// TwinCAT 3 PLC project main
// ProgramVersion: 3.1.4024.0
// libraries:
//   Tc2_Standard, * (Beckhoff Automation GmbH)
//   Tc2_System, * (Beckhoff Automation GmbH)
//   Tc3_Module, * (Beckhoff Automation GmbH)
// project tree:
//   DUTs/ SafeState.TcDUT
//   GVLs/ IO.TcGVL
//   / PlcTask.TcTTO
//   POUs/ FB_EdgeDetector.TcPOU, MAIN.TcPOU
// real-time tasks:
//   TASK PlcTask: cycle T#10ms, priority 20, ADS port 350
// I/O:
//   DEVICE Device 1 (EtherCAT), AmsNetId 10.180.42.11.2.1
//     Term 1 (EK1200) [EK1200-5000 EtherCAT Power supply (2A E-Bus)]
//       Term 2 (EL1004) [EL1004 4Ch. Dig. Input 24V, 3ms]
//       Term 3 (EL2004) [EL2004 4Ch. Dig. Output 24V, 0.5A]
//       Term 4 (EL3004) [EL3004 4Ch. Ana. Input +/-10V]
//       Term 5 (EL4034) [EL4034 4Ch. Ana. Output +/-10V, 12bit]
//       Term 6 (EK1110) [EK1110 EtherCAT extension]
// variable links:
//   main/main Instance <-> Device 1 (EtherCAT)/Term 1 (EK1200)/Term 2 (EL1004)
//     PlcTask Inputs/IO.bBlueButton <-> Channel 2/Input
//     PlcTask Inputs/IO.bYellowButton <-> Channel 1/Input
//   main/main Instance <-> Device 1 (EtherCAT)/Term 1 (EK1200)/Term 3 (EL2004)
//     PlcTask Outputs/IO.bGreenLight <-> Channel 2/Output
//     PlcTask Outputs/IO.bRedLight <-> Channel 1/Output

CONFIGURATION main
    RESOURCE PLC ON TwinCAT3
        TASK PlcTask(INTERVAL := T#10ms, PRIORITY := 20);
        PROGRAM MAIN WITH PlcTask : MAIN;
    END_RESOURCE
END_CONFIGURATION

// ---- DUTs/SafeState.TcDUT
{attribute 'qualified_only'}
{attribute 'strict'}
TYPE SafeState :
(
	Init := 0,
	Close,
	CheckDigit,
	Open,
	WrongCode
);
END_TYPE

// ---- GVLs/IO.TcGVL
{attribute 'qualified_only'}
VAR_GLOBAL
	bYellowButton 	AT %I*:BOOL;
	bBlueButton		AT %I* :BOOL;
	
	bGreenLight		AT %Q*:BOOL;
	bRedLight		AT %Q*:BOOL;
	
	iUltraschallSensor AT %I*:INT;
END_VAR

// ---- POUs/MAIN.TcPOU
PROGRAM MAIN
VAR
	actualState	:		SafeState := SafeState.Init;	

	blueEdgeDetector : 		FB_EdgeDetector;
	yellowEdgeDetector :	FB_EdgeDetector;
	codeArray : 			ARRAY[0..3] OF BOOL;  // Array mit 4 Elementen vom Typ BOOL
	currentIndex :			INT := 0;
	correctIndex :			INT := 0;
	timer :					TON;
END_VAR

VAR CONSTANT
    lightDuration : TIME := T#5S;
END_VAR

blueEdgeDetector(inputValue:=IO.bBlueButton,DoublePressedTime := 10);
yellowEdgeDetector(inputValue:=IO.bYellowButton,DoublePressedTime := 10);


CASE actualState OF
	SafeState.Init:
	IF NOT(blueEdgeDetector.risingEdge = TRUE AND yellowEdgeDetector.risingEdge = TRUE) THEN
		IF blueEdgeDetector.risingEdge = TRUE THEN
			codeArray[currentIndex] := TRUE;
			currentIndex := currentIndex + 1;
		ELSE
			IF yellowEdgeDetector.risingEdge = TRUE THEN
				codeArray[currentIndex] := FALSE;
				currentIndex := currentIndex + 1;
			END_IF
		END_IF
		IF currentIndex >= 4 THEN
			actualState := SafeState.Close;
			currentIndex := 0;
		END_IF
	END_IF
	;
	SafeState.Close:
		timer(IN:= FALSE,PT:=lightDuration);
		IO.bGreenLight := FALSE;
		IO.bRedLight := FALSE;
		actualState := SafeState.CheckDigit;
	;
	SafeState.CheckDigit:
	IF NOT(blueEdgeDetector.risingEdge = TRUE AND yellowEdgeDetector.risingEdge = TRUE) THEN
		IF blueEdgeDetector.risingEdge = TRUE THEN
			IF codeArray[currentIndex] = TRUE THEN
				correctIndex := correctIndex + 1;
			END_IF
			currentIndex := currentIndex + 1;
		ELSE
			IF yellowEdgeDetector.risingEdge = TRUE THEN
				IF codeArray[currentIndex] = FALSE THEN
					correctIndex := correctIndex + 1;
				END_IF
				currentIndex := currentIndex + 1;
			END_IF
		END_IF

		IF currentIndex >= 4 THEN
			currentIndex := 0;
			IF correctIndex >= 4 THEN
				correctIndex:= 0;
				actualState := SafeState.Open;
			ELSE
				correctIndex := 0;
				actualState := SafeState.WrongCode;
			END_IF
		END_IF
	END_IF
	;
	SafeState.Open:
	IO.bGreenLight := TRUE;
	timer(IN:= TRUE,PT:=lightDuration);
	IF timer.Q = TRUE THEN
		actualState := SafeState.Close;
	END_IF
	;
	SafeState.WrongCode:
	IO.bRedLight := TRUE;
	timer(IN:= TRUE,PT:=lightDuration);
	IF timer.Q = TRUE THEN
		actualState := SafeState.Close;
	END_IF
	;
END_CASE

END_PROGRAM

// ---- POUs/FB_EdgeDetector.TcPOU
FUNCTION_BLOCK FB_EdgeDetector
VAR_INPUT
	inputValue : BOOL;
	DoublePressedTime: UINT;
END_VAR
VAR_OUTPUT
	risingEdge : BOOL;
	fallingEdge : BOOL;
	DoublePressed: BOOL;
END_VAR
VAR
	inputValue_old : BOOL;
	OncePressed: BOOL := FALSE;
	DoublePressedcounter: UINT := 0;
END_VAR

risingEdge := FALSE;
fallingEdge := FALSE;
DoublePressed := FALSE;

IF inputValue <> inputValue_old THEN
	IF inputValue = TRUE THEN
		risingEdge := TRUE;
		IF OncePressed = FALSE THEN
			OncePressed := TRUE;
		ELSE
			OncePressed := FALSE;
			DoublePressed := TRUE;
			DoublePressedcounter := 0;
		END_IF
	ELSE
		fallingEdge := TRUE;
	END_IF
END_IF
inputValue_old := inputValue;
IF OncePressed = TRUE THEN
	IF DoublePressedcounter >= DoublePressedTime THEN
		OncePressed := FALSE;
		DoublePressedcounter := 0;
	ELSE
		DoublePressedcounter := DoublePressedcounter + 1;
	END_IF	
END_IF

END_FUNCTION_BLOCK
